// TIA Portal V20 export
TYPE "typeEm7Monitoring"
// stored: Access Published, Namespace Unit1
   STRUCT
      jobinterface { ExternalWritable := 'False'} : "Unit1.typeEm7MonitoringJobInterface";
      jobWorkingDone { ExternalWritable := 'False'} : "Unit1.typeEm7MonitoringJobWorkingDone";
      jobStatus { ExternalWritable := 'False'} : "Unit1.typeEm7MonitoringJobStatus";
      cmStatus { ExternalWritable := 'False'} : "Unit1.typeEm7MonitoringCmStatus";
      UserDefine { ExternalWritable := 'False'} : "Unit1.typeEm7MonitoringUserDefine";
   END_STRUCT;
END_TYPE
